RoboDK station: Station.rdk

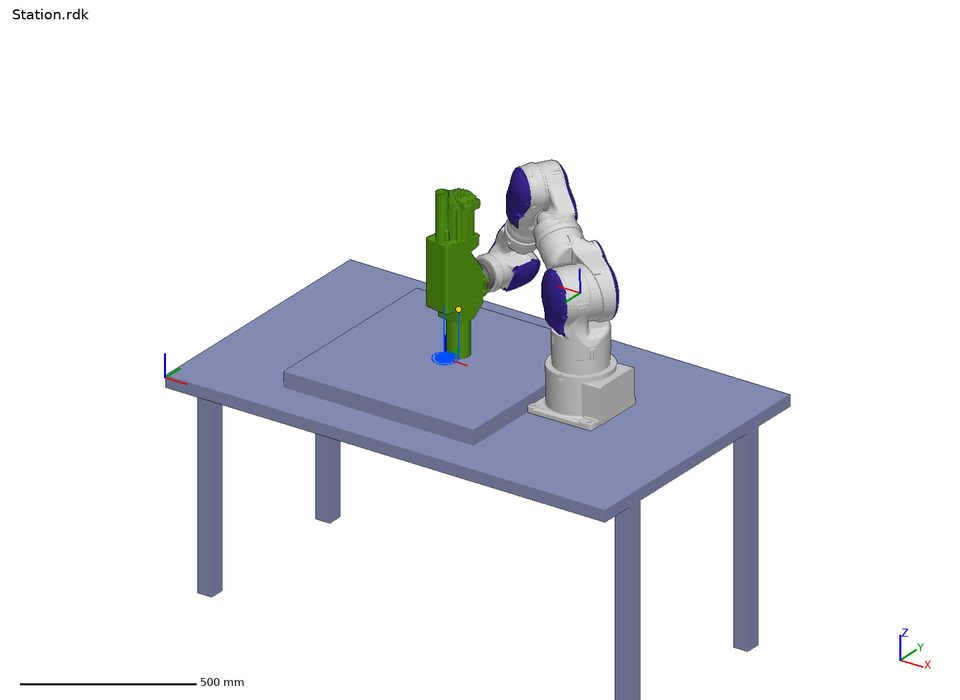
[picture v0: the station drawn from its stored meshes, robots at their saved joint values, targets as dots, program paths as lines]
Station Station (saved by RoboDK 5.5.3). Poses are relative to the parent item; angles as X-Y-Z fixed-axis rotations.
Station parameters (name, value as stored): Balls, 9000, lastSpeed, 40.0, LASTSPEED, 40.0
  - frame Yaskawa SIA10D Base at (1117.6, 457, 397.69) mm, rotated rx 0 ry 0.65 rz -180 deg
    - robot Yaskawa SIA10D: 7 axes, payload 10 kg, reach 720 mm, repeatability 0.1 mm, weight 60 kg
        modified DH rows (alpha deg, a mm, theta deg, d mm): 0, 0, 0, 360; -90, 0, 0, 0; 90, 0, 0, 360; -90, 0, 0, 0; 90, 0, 0, 360; -90, 0, 0, 0; 90, 0, 180, 155
        base shift (0, 0, -360) mm
        joint limits [-180, -110, -170, -135, -180, -110, -180] to [180, 110, 170, 135, 180, 110, 180]; home [0, 0, 0, 90, 0, 0, 0]; saved at [-31.519, 54.462, 0, 96.238, 71.076, 100.442, -153.064]
      - tool MDPH2, TCP at (-228, 0, 70.1) mm, rotated rx 0 ry -90 rz 0 deg, size 541.9 x 124.6 x 162.8 mm, geometry from Working one.STEP
  - frame Printing Frame at (649.7, 457, 58.96) mm
    - object par3 at (0, 0, 0) mm, rotated rx 90 ry 0 rz 0 deg, size 59.1 x 2 x 60 mm, geometry from par3.STEP
  - machining project Print3D settings: C:/Users/ajh269/AppData/Local/Temp/par2.stl | rotZ(0) | rotX(0)*rotY(0) | rotz(0)
  - Python program MCodeHandler (listed below)
  - Python program onStart (listed below)
  - Python program ExtruderHandler (listed below)
  - object table at (0, 0, -30) mm, rotated rx 90 ry 0 rz 0 deg, size 1524 x 739.1 x 914.4 mm, geometry from table.STEP
  - frame Table Corner at (0, 0, 0) mm
  - object MD_Bed at (320.1, 127, 5.56) mm, rotated rx 90 ry 0 rz 180 deg, size 660 x 53.3 x 660 mm, geometry from MD_Bed.STEP
  - machining project Print3D settings: C:/Users/ajh269/AppData/Local/Temp/par3.stl | rotZ(0) | rotX(0)*rotY(0) | rotz(0) | onStart | onPathStart | onApproach | onPoint | onRetract | onFinish | SetRPM(%1) | SetTool(%1) | ExtruderHandler(%1) | default | default | OutOnMov(%1) | OutOffMov(%1) | onPathFinish | MCodeHandler(%1)
  - program Print3D (604 instructions, listed below)
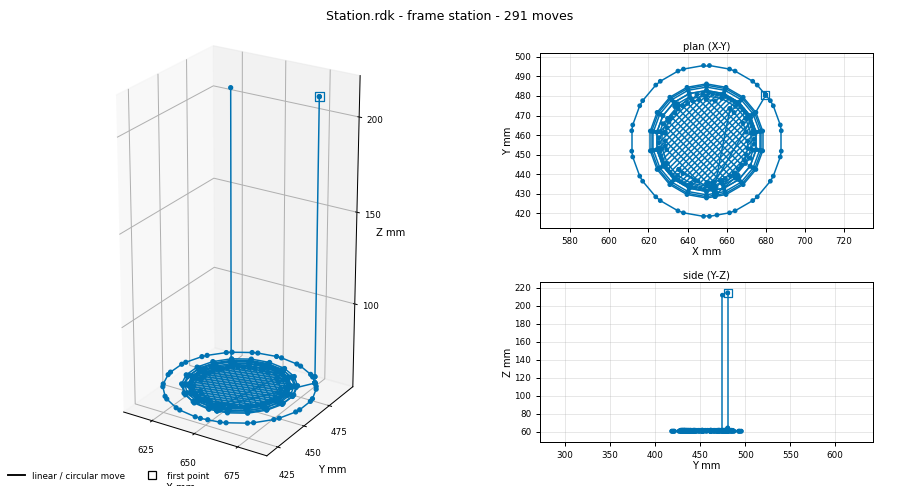
[picture p0: tool path of Station.rdk in frame station, 291 of 291 moves have a stored position in this frame; points joined in program order, loops and branches not executed]

--- Python program MCodeHandler ---
import sys

def handleFanOn():
    pass

def handleFanOff():
    pass

def handleTemperatureAsync():
    pass

def handleTemperatureSync():
    pass

# Create a mapping for the instruction codes
callbacks = {
    106: handleFanOn,
    107: handleFanOff,
    104: handleTemperatureAsync,
    109: handleTemperatureSync,
}

if len(sys.argv) > 1:
    instructionCode = int(sys.argv[1])
    print(instructionCode)

    if(len(sys.argv) > 2):
        arg = float(sys.argv[2])
        print(arg)

    #check for a second argument depending on the first

# Provoking an exception will display the console output if you run this script from RoboDK
# raise Exception('Display output. If program was run accidentally, move the error message above the pause button on RoboDK and click fast. (Shortcut is Backspace)')

--- Python program onStart ---
# import serial

# ser = serial.Serial('COM6', 9600, timeout=1.0)

# ser.write(b"NEW_PRINT\n")
# print(ser.readline())

--- Python program ExtruderHandler ---
# Type help("robodk.robolink") or help("robodk.robomath") for more information
# Press F5 to run the script
# Documentation: https://robodk.com/doc/en/RoboDK-API.html
# Reference:     https://robodk.com/doc/en/PythonAPI/robodk.html
# Note: It is not required to keep a copy of this file, your Python script is saved with your RDK project

# You can also use the new version of the API:
# from robodk import robolink    # RoboDK API
# from robodk import robomath    # Robot toolbox
# RDK = robolink.Robolink()

# Forward and backwards compatible use of the RoboDK API:
# Remove these 2 lines to follow python programming guidelines
# from robodk import *      # RoboDK API
# from robolink import *    # Robot toolbox
# Link to RoboDK
# RDK = Robolink()

import socket

message = b'{ distance: %f, materialLength: %f, newSpeed: %f }' % (1, 1, 0)

UDP_IP = "10.0.0.111"
UDP_PORT = 8888

sock = socket.socket(socket.AF_INET, # Internet
                    socket.SOCK_DGRAM) # UDP
sock.sendto(message, (UDP_IP, UDP_PORT))

# Provoking an exception will display the console output if you run this script from RoboDK
# raise Exception('Display output. If program was run accidentally, move the error message above the pause button on RoboDK and click fast. (Shortcut is Backspace)')

--- program Print3D (robot Yaskawa SIA10D) ---
  Smooth(1)
  Call MCodeHandler(107)
  Call MCodeHandler(104)
  Set speed (83.3 mm/s)
  Set Ref.: Printing Frame
  Set Tool: MDPH2
  Show MDPH2
  MoveJ 1 to (30.12, 23.57, 155) mm, rotated rx 180 ry 0 rz -100 deg; joints [-31.631, 34.814, 0, 98.46, 74.874, 105.649, -135.983]
  MoveL 2 to (30.12, 23.57, 155) mm, rotated rx 180 ry 0 rz -100 deg; joints [-31.631, 34.814, 0, 98.46, 74.874, 105.649, -135.983]
  MoveL 3 to (30.12, 23.57, 5) mm, rotated rx 180 ry 0 rz -100 deg; joints [-31.522, 53.972, 0, 96.405, 71.131, 100.548, -152.753]
  MoveL 4 to (30.12, 23.57, 5) mm, rotated rx 180 ry 0 rz -100 deg; joints [-31.522, 53.972, 0, 96.405, 71.131, 100.548, -152.753]
  Call MCodeHandler(109)
  Call MCodeHandler(83)
  Set speed (130.0 mm/s)
  MoveL 5 to (30.12, 23.57, 1.5) mm, rotated rx 180 ry 0 rz -100 deg; joints [-31.519, 54.462, 0, 96.238, 71.076, 100.442, -153.064]
  Call ExtruderHandler(-14.137...: ExtruderHandler(-14.13717)
  Set speed (40.0 mm/s)
  MoveL 6 to (30.12, 23.57, 1.5) mm, rotated rx 180 ry 0 rz -100 deg; joints [-31.519, 54.462, 0, 96.238, 71.076, 100.442, -153.064]
  Set speed (130.0 mm/s)
  MoveL 7 to (30.12, 23.57, 1.5) mm, rotated rx 180 ry 0 rz -100 deg; joints [-31.519, 54.462, 0, 96.238, 71.076, 100.442, -153.064]
  Call ExtruderHandler(14.13717)
  Set speed (40.0 mm/s)
  MoveL 8 to (30.12, 23.57, 1.5) mm, rotated rx 180 ry 0 rz -100 deg; joints [-31.519, 54.462, 0, 96.238, 71.076, 100.442, -153.064]
  Set speed (30.0 mm/s)
  MoveL 9 to (30.12, 23.57, 1.5) mm, rotated rx 180 ry 0 rz -100 deg; joints [-31.519, 54.462, 0, 96.238, 71.076, 100.442, -153.064]
  Call ExtruderHandler(26.15888)
  MoveL 10 to (25.93, 28.56, 1.5) mm, rotated rx -180 ry 0 rz -100 deg; joints [-31.768, 54.946, 0, 94.943, 70.997, 100.822, -152.324]
  Call ExtruderHandler(12.10715)
  MoveL 11 to (23.62, 30.5, 1.5) mm, rotated rx -180 ry 0 rz -100 deg; joints [-31.82, 55.182, 0, 94.314, 71.022, 100.974, -151.954]
  Call ExtruderHandler(41.85421)
  MoveL 12 to (14.6, 35.71, 1.5) mm, rotated rx -180 ry 0 rz -100 deg; joints [-31.781, 56.028, 0, 92.089, 71.315, 101.401, -150.617]
  Call ExtruderHandler(12.10718)
  MoveL 13 to (11.77, 36.74, 1.5) mm, rotated rx -180 ry 0 rz -100 deg; joints [-31.71, 56.273, 0, 91.451, 71.453, 101.49, -150.225]
  Call ExtruderHandler(41.85419)
  MoveL 14 to (1.51, 38.55, 1.5) mm, rotated rx 180 ry 0 rz -100 deg; joints [-31.269, 57.096, 0, 89.328, 72.091, 101.669, -148.889]
  Call ExtruderHandler(12.10714)
  MoveL 15 to (-1.51, 38.55, 1.5) mm, rotated rx 180 ry 0 rz -100 deg; joints [-31.091, 57.32, 0, 88.757, 72.314, 101.681, -148.519]
  Call ExtruderHandler(41.85422)
  MoveL 16 to (-11.77, 36.74, 1.5) mm, rotated rx -180 ry 0 rz -100 deg; joints [-30.325, 58.016, 0, 86.988, 73.183, 101.585, -147.342]
  Call ExtruderHandler(12.10717)
  MoveL 17 to (-14.6, 35.71, 1.5) mm, rotated rx -180 ry 0 rz -100 deg; joints [-30.066, 58.189, 0, 86.551, 73.455, 101.518, -147.041]
  Call ExtruderHandler(41.85421)
  MoveL 18 to (-23.62, 30.5, 1.5) mm, rotated rx 180 ry 0 rz -100 deg; joints [-29.069, 58.666, 0, 85.348, 74.438, 101.161, -146.165]
  Call ExtruderHandler(12.10715)
  MoveL 19 to (-25.93, 28.56, 1.5) mm, rotated rx 180 ry 0 rz -100 deg; joints [-28.759, 58.765, 0, 85.099, 74.726, 101.025, -145.968]
  Call ExtruderHandler(41.85420)
  MoveL 20 to (-32.63, 20.58, 1.5) mm, rotated rx 180 ry 0 rz -100 deg; joints [-27.638, 58.956, 0, 84.61, 75.717, 100.46, -145.503]
  Call ExtruderHandler(12.10718)
  MoveL 21 to (-34.14, 17.97, 1.5) mm, rotated rx 180 ry 0 rz -100 deg; joints [-27.308, 58.967, 0, 84.58, 75.995, 100.274, -145.435]
  Call ExtruderHandler(41.85421)
  MoveL 22 to (-37.7, 8.18, 1.5) mm, rotated rx 180 ry 0 rz -100 deg; joints [-26.172, 58.846, 0, 84.865, 76.909, 99.581, -145.437]
  Call ExtruderHandler(12.10715)
  MoveL 23 to (-38.22, 5.21, 1.5) mm, rotated rx -180 ry 0 rz -100 deg; joints [-25.853, 58.766, 0, 85.058, 77.155, 99.372, -145.506]
  Call ExtruderHandler(41.85420)
  MoveL 24 to (-38.22, -5.21, 1.5) mm, rotated rx -180 ry 0 rz -100 deg; joints [-24.811, 58.349, 0, 86.082, 77.926, 98.645, -145.973]
  Call ExtruderHandler(12.10715)
  MoveL 25 to (-37.7, -8.18, 1.5) mm, rotated rx 180 ry 0 rz -100 deg; joints [-24.535, 58.192, 0, 86.473, 78.121, 98.44, -146.17]
  Call ExtruderHandler(41.85422)
  MoveL 26 to (-34.14, -17.97, 1.5) mm, rotated rx 180 ry 0 rz -100 deg; joints [-23.696, 57.537, 0, 88.11, 78.687, 97.773, -147.044]
  Call ExtruderHandler(12.10716)
  MoveL 27 to (-32.63, -20.58, 1.5) mm, rotated rx -180 ry 0 rz -100 deg; joints [-23.493, 57.322, 0, 88.651, 78.814, 97.597, -147.345]
  Call ExtruderHandler(41.85420)
  MoveL 28 to (-25.93, -28.56, 1.5) mm, rotated rx -180 ry 0 rz -80 deg; joints [-19.878, 63.594, 0, 73.405, 67.135, 109.774, -141.706]
  Call ExtruderHandler(12.10716)
  MoveL 29 to (-23.62, -30.5, 1.5) mm, rotated rx 180 ry 0 rz -80 deg; joints [-19.773, 63.278, 0, 74.141, 67.083, 109.544, -142.089]
  Call ExtruderHandler(41.85421)
  MoveL 30 to (-14.6, -35.71, 1.5) mm, rotated rx 180 ry 0 rz -80 deg; joints [-19.582, 62.167, 0, 76.758, 66.761, 108.837, -143.502]
  Call ExtruderHandler(12.10716)
  MoveL 31 to (-11.77, -36.74, 1.5) mm, rotated rx 180 ry 0 rz -80 deg; joints [-19.58, 61.849, 0, 77.513, 66.626, 108.662, -143.926]
  Call ExtruderHandler(41.85420)
  MoveL 32 to (-1.51, -38.55, 1.5) mm, rotated rx -180 ry 0 rz -80 deg; joints [-19.763, 60.795, 0, 80.039, 66.021, 108.179, -145.395]
  Call ExtruderHandler(12.10714)
  MoveL 33 to (1.51, -38.55, 1.5) mm, rotated rx 180 ry 0 rz -80 deg; joints [-19.872, 60.511, 0, 80.724, 65.808, 108.078, -145.811]
  Call ExtruderHandler(15.69532)
  MoveL 34 to (5.36, -37.87, 1.5) mm, rotated rx -180 ry 0 rz -80 deg; joints [-20.08, 60.177, 0, 81.535, 65.486, 107.999, -146.324]
  Call ExtruderHandler(26.15890)
  MoveL 35 to (11.77, -36.74, 1.5) mm, rotated rx 180 ry 0 rz -80 deg; joints [-20.433, 59.631, 0, 82.869, 64.946, 107.866, -147.171]
  Call ExtruderHandler(12.10714)
  MoveL 36 to (14.6, -35.71, 1.5) mm, rotated rx 180 ry 0 rz -80 deg; joints [-20.645, 59.413, 0, 83.406, 64.667, 107.846, -147.532]
  Call ExtruderHandler(41.85423)
  MoveL 37 to (23.62, -30.5, 1.5) mm, rotated rx 180 ry 0 rz -80 deg; joints [-21.531, 58.8, 0, 84.926, 63.619, 107.928, -148.632]
  Call ExtruderHandler(12.10716)
  MoveL 38 to (25.93, -28.56, 1.5) mm, rotated rx 180 ry 0 rz -80 deg; joints [-21.823, 58.668, 0, 85.255, 63.301, 107.994, -148.899]
  Call ExtruderHandler(41.85420)
  MoveL 39 to (32.63, -20.58, 1.5) mm, rotated rx 180 ry 0 rz -80 deg; joints [-22.922, 58.383, 0, 85.976, 62.186, 108.366, -149.617]
  Call ExtruderHandler(12.10714)
  MoveL 40 to (34.14, -17.97, 1.5) mm, rotated rx -180 ry 0 rz -80 deg; joints [-23.254, 58.352, 0, 86.058, 61.871, 108.513, -149.76]
  Call ExtruderHandler(41.85421)
  MoveL 41 to (37.7, -8.18, 1.5) mm, rotated rx 180 ry 0 rz -80 deg; joints [-24.408, 58.422, 0, 85.897, 60.851, 109.147, -150.015]
  Call ExtruderHandler(12.10718)
  MoveL 42 to (38.22, -5.21, 1.5) mm, rotated rx 180 ry 0 rz -80 deg; joints [-24.731, 58.493, 0, 85.723, 60.588, 109.362, -150.018]
  Call ExtruderHandler(41.85420)
  MoveL 43 to (38.22, 5.21, 1.5) mm, rotated rx -180 ry 0 rz -100 deg; joints [-30.075, 53.231, 0, 99.601, 72.038, 99.119, -154.896]
  Call ExtruderHandler(12.10718)
  MoveL 44 to (37.7, 8.18, 1.5) mm, rotated rx 180 ry 0 rz -100 deg; joints [-30.365, 53.375, 0, 99.205, 71.812, 99.324, -154.695]
  Call ExtruderHandler(41.85422)
  MoveL 45 to (34.14, 17.97, 1.5) mm, rotated rx -180 ry 0 rz -100 deg; joints [-31.188, 53.977, 0, 97.553, 71.234, 100.022, -153.809]
  Call ExtruderHandler(12.10713)
  MoveL 46 to (32.63, 20.58, 1.5) mm, rotated rx 180 ry 0 rz -100 deg; joints [-31.367, 54.178, 0, 97.007, 71.131, 100.215, -153.506]
  Call ExtruderHandler(14.79146)
  MoveL 47 to (30.26, 23.4, 1.5) mm, rotated rx 180 ry 0 rz -100 deg; joints [-31.511, 54.446, 0, 96.282, 71.079, 100.429, -153.089]
  Call ExtruderHandler(-14.137...: ExtruderHandler(-14.13717)
  Set speed (40.0 mm/s)
  MoveL 48 to (30.26, 23.4, 1.5) mm, rotated rx 180 ry 0 rz -100 deg; joints [-31.511, 54.446, 0, 96.282, 71.079, 100.429, -153.089]
  Set speed (130.0 mm/s)
  MoveL 49 to (3.4, -22.44, 1.5) mm, rotated rx -180 ry 0 rz -80 deg; joints [-21.539, 60.913, 0, 79.77, 64.533, 109.262, -145.748]
  Call ExtruderHandler(14.13717)
  Set speed (40.0 mm/s)
  MoveL 50 to (3.4, -22.44, 1.5) mm, rotated rx -180 ry 0 rz -80 deg; joints [-21.539, 60.913, 0, 79.77, 64.533, 109.262, -145.748]
  Set speed (30.0 mm/s)
  MoveL 51 to (3.4, -22.44, 1.5) mm, rotated rx -180 ry 0 rz -80 deg; joints [-21.539, 60.913, 0, 79.77, 64.533, 109.262, -145.748]
  Call ExtruderHandler(18.28870)
  MoveL 52 to (7.88, -21.65, 1.5) mm, rotated rx -180 ry 0 rz -80 deg; joints [-21.792, 60.526, 0, 80.708, 64.139, 109.168, -146.346]
  Call ExtruderHandler(32.14129)
  MoveL 53 to (14.81, -17.65, 1.5) mm, rotated rx 180 ry 0 rz -80 deg; joints [-22.467, 60.044, 0, 81.882, 63.33, 109.237, -147.2]
  Call ExtruderHandler(32.14129)
  MoveL 54 to (19.95, -11.52, 1.5) mm, rotated rx 180 ry 0 rz -80 deg; joints [-23.289, 59.819, 0, 82.44, 62.496, 109.536, -147.758]
  Call ExtruderHandler(32.14130)
  MoveL 55 to (22.69, -4, 1.5) mm, rotated rx 180 ry 0 rz -100 deg; joints [-28.12, 53.888, 0, 97.749, 73.988, 98.597, -153.471]
  Call ExtruderHandler(32.14128)
  MoveL 56 to (22.69, 4, 1.5) mm, rotated rx 180 ry 0 rz -100 deg; joints [-28.988, 54.182, 0, 96.958, 73.281, 99.136, -153.107]
  Call ExtruderHandler(32.14131)
  MoveL 57 to (19.95, 11.52, 1.5) mm, rotated rx 180 ry 0 rz -100 deg; joints [-29.626, 54.653, 0, 95.695, 72.836, 99.665, -152.43]
  Call ExtruderHandler(32.14129)
  MoveL 58 to (14.81, 17.65, 1.5) mm, rotated rx 180 ry 0 rz -100 deg; joints [-29.959, 55.247, 0, 94.113, 72.703, 100.117, -151.523]
  Call ExtruderHandler(32.14130)
  MoveL 59 to (7.88, 21.65, 1.5) mm, rotated rx 180 ry 0 rz -100 deg; joints [-29.96, 55.897, 0, 92.405, 72.886, 100.431, -150.495]
  Call ExtruderHandler(32.14128)
  MoveL 60 to (0, 23.04, 1.5) mm, rotated rx 180 ry 0 rz -100 deg; joints [-29.643, 56.523, 0, 90.774, 73.341, 100.561, -149.468]
  Call ExtruderHandler(32.14129)
  MoveL 61 to (-7.88, 21.65, 1.5) mm, rotated rx 180 ry 0 rz -100 deg; joints [-29.06, 57.049, 0, 89.417, 73.995, 100.489, -148.566]
  Call ExtruderHandler(32.14130)
  MoveL 62 to (-14.81, 17.65, 1.5) mm, rotated rx 180 ry 0 rz -100 deg; joints [-28.281, 57.407, 0, 88.495, 74.762, 100.224, -147.895]
  Call ExtruderHandler(32.14129)
  MoveL 63 to (-19.95, 11.52, 1.5) mm, rotated rx 180 ry 0 rz -100 deg; joints [-27.395, 57.551, 0, 88.12, 75.556, 99.801, -147.539]
  Call ExtruderHandler(32.14129)
  MoveL 64 to (-22.69, 4, 1.5) mm, rotated rx 180 ry 0 rz -100 deg; joints [-26.497, 57.46, 0, 88.339, 76.299, 99.28, -147.539]
  Call ExtruderHandler(32.14129)
  MoveL 65 to (-22.69, -4, 1.5) mm, rotated rx -180 ry 0 rz -100 deg; joints [-25.68, 57.147, 0, 89.123, 76.921, 98.726, -147.896]
  Call ExtruderHandler(32.14129)
  MoveL 66 to (-19.95, -11.52, 1.5) mm, rotated rx -180 ry 0 rz -100 deg; joints [-25.035, 56.653, 0, 90.378, 77.361, 98.211, -148.567]
  Call ExtruderHandler(32.14129)
  MoveL 67 to (-14.81, -17.65, 1.5) mm, rotated rx -180 ry 0 rz -100 deg; joints [-24.64, 56.041, 0, 91.955, 77.568, 97.795, -149.472]
  Call ExtruderHandler(32.14130)
  MoveL 68 to (-7.88, -21.65, 1.5) mm, rotated rx -180 ry 0 rz -80 deg; joints [-21.186, 62.026, 0, 77.108, 65.333, 109.713, -144.157]
  Call ExtruderHandler(32.14129)
  MoveL 69 to (0, -23.04, 1.5) mm, rotated rx 180 ry 0 rz -80 deg; joints [-21.349, 61.212, 0, 79.052, 64.83, 109.333, -145.291]
  Call ExtruderHandler(12.94872)
  MoveL 70 to (3.17, -22.48, 1.5) mm, rotated rx 180 ry 0 rz -80 deg; joints [-21.526, 60.933, 0, 79.723, 64.552, 109.267, -145.718]
  Call ExtruderHandler(-14.137...: ExtruderHandler(-14.13717)
  Set speed (40.0 mm/s)
  MoveL 71 to (3.17, -22.48, 1.5) mm, rotated rx 180 ry 0 rz -80 deg; joints [-21.526, 60.933, 0, 79.723, 64.552, 109.267, -145.718]
  Set speed (130.0 mm/s)
  MoveL 72 to (3.86, -25.08, 1.5) mm, rotated rx 180 ry 0 rz -80 deg; joints [-21.297, 60.771, 0, 80.11, 64.681, 109.04, -145.867]
  Call ExtruderHandler(14.13717)
  Set speed (40.0 mm/s)
  MoveL 73 to (3.86, -25.08, 1.5) mm, rotated rx 180 ry 0 rz -80 deg; joints [-21.297, 60.771, 0, 80.11, 64.681, 109.04, -145.867]
  Set speed (30.0 mm/s)
  MoveL 74 to (3.86, -25.08, 1.5) mm, rotated rx 180 ry 0 rz -80 deg; joints [-21.297, 60.771, 0, 80.11, 64.681, 109.04, -145.867]
  Call ExtruderHandler(20.18568)
  MoveL 75 to (8.81, -24.2, 1.5) mm, rotated rx 180 ry 0 rz -80 deg; joints [-21.576, 60.345, 0, 81.143, 64.249, 108.936, -146.526]
  Call ExtruderHandler(35.93525)
  MoveL 76 to (16.56, -19.73, 1.5) mm, rotated rx 180 ry 0 rz -80 deg; joints [-22.331, 59.809, 0, 82.454, 63.345, 109.012, -147.479]
  Call ExtruderHandler(35.93525)
  MoveL 77 to (22.31, -12.88, 1.5) mm, rotated rx 180 ry 0 rz -80 deg; joints [-23.255, 59.558, 0, 83.076, 62.409, 109.343, -148.101]
  Call ExtruderHandler(35.93526)
  MoveL 78 to (25.37, -4.47, 1.5) mm, rotated rx 180 ry 0 rz -80 deg; joints [-24.221, 59.62, 0, 82.937, 61.567, 109.898, -148.321]
  Call ExtruderHandler(35.93524)
  MoveL 79 to (25.37, 4.47, 1.5) mm, rotated rx -180 ry 0 rz -100 deg; joints [-29.2, 54.024, 0, 97.394, 73.049, 99.153, -153.405]
  Call ExtruderHandler(35.93527)
  MoveL 80 to (22.31, 12.88, 1.5) mm, rotated rx 180 ry 0 rz -100 deg; joints [-29.912, 54.548, 0, 95.98, 72.55, 99.746, -152.648]
  Call ExtruderHandler(35.93524)
  MoveL 81 to (16.56, 19.73, 1.5) mm, rotated rx 180 ry 0 rz -100 deg; joints [-30.279, 55.212, 0, 94.212, 72.408, 100.254, -151.634]
  Call ExtruderHandler(35.93526)
  MoveL 82 to (8.81, 24.2, 1.5) mm, rotated rx 180 ry 0 rz -100 deg; joints [-30.274, 55.938, 0, 92.301, 72.62, 100.607, -150.485]
  Call ExtruderHandler(35.93524)
  MoveL 83 to (0, 25.76, 1.5) mm, rotated rx 180 ry 0 rz -100 deg; joints [-29.916, 56.64, 0, 90.478, 73.136, 100.754, -149.337]
  Call ExtruderHandler(35.93524)
  MoveL 84 to (-8.81, 24.2, 1.5) mm, rotated rx 180 ry 0 rz -100 deg; joints [-29.263, 57.229, 0, 88.96, 73.87, 100.673, -148.327]
  Call ExtruderHandler(35.93526)
  MoveL 85 to (-16.56, 19.73, 1.5) mm, rotated rx 180 ry 0 rz -100 deg; joints [-28.395, 57.631, 0, 87.93, 74.725, 100.375, -147.578]
  Call ExtruderHandler(35.93525)
  MoveL 86 to (-22.31, 12.88, 1.5) mm, rotated rx 180 ry 0 rz -100 deg; joints [-27.409, 57.792, 0, 87.511, 75.606, 99.901, -147.179]
  Call ExtruderHandler(35.93525)
  MoveL 87 to (-25.37, 4.47, 1.5) mm, rotated rx 180 ry 0 rz -100 deg; joints [-26.41, 57.69, 0, 87.755, 76.429, 99.315, -147.18]
  Call ExtruderHandler(35.93525)
  MoveL 88 to (-25.37, -4.47, 1.5) mm, rotated rx 180 ry 0 rz -100 deg; joints [-25.5, 57.339, 0, 88.632, 77.118, 98.696, -147.579]
  Call ExtruderHandler(35.93525)
  MoveL 89 to (-22.31, -12.88, 1.5) mm, rotated rx 180 ry 0 rz -100 deg; joints [-24.779, 56.785, 0, 90.036, 77.609, 98.12, -148.329]
  Call ExtruderHandler(35.93525)
  MoveL 90 to (-16.56, -19.73, 1.5) mm, rotated rx 180 ry 0 rz -100 deg; joints [-24.333, 56.1, 0, 91.798, 77.846, 97.657, -149.34]
  Call ExtruderHandler(35.93526)
  MoveL 91 to (-8.81, -24.2, 1.5) mm, rotated rx -180 ry 0 rz -80 deg; joints [-20.905, 62.02, 0, 77.121, 65.571, 109.543, -144.082]
  Call ExtruderHandler(35.93525)
  MoveL 92 to (0, -25.76, 1.5) mm, rotated rx 180 ry 0 rz -80 deg; joints [-21.083, 61.11, 0, 79.293, 65.016, 109.12, -145.349]
  Call ExtruderHandler(14.84570)
  MoveL 93 to (3.64, -25.12, 1.5) mm, rotated rx 180 ry 0 rz -80 deg; joints [-21.285, 60.791, 0, 80.063, 64.7, 109.044, -145.837]
  Call ExtruderHandler(-14.137...: ExtruderHandler(-14.13717)
  Set speed (40.0 mm/s)
  MoveL 94 to (3.64, -25.12, 1.5) mm, rotated rx 180 ry 0 rz -80 deg; joints [-21.285, 60.791, 0, 80.063, 64.7, 109.044, -145.837]
  Set speed (130.0 mm/s)
  MoveL 95 to (4.33, -27.71, 1.5) mm, rotated rx -180 ry 0 rz -80 deg; joints [-21.054, 60.631, 0, 80.446, 64.831, 108.818, -145.985]
  Call ExtruderHandler(14.13717)
  Set speed (40.0 mm/s)
  MoveL 96 to (4.33, -27.71, 1.5) mm, rotated rx -180 ry 0 rz -80 deg; joints [-21.054, 60.631, 0, 80.446, 64.831, 108.818, -145.985]
  Set speed (30.0 mm/s)
  MoveL 97 to (4.33, -27.71, 1.5) mm, rotated rx -180 ry 0 rz -80 deg; joints [-21.054, 60.631, 0, 80.446, 64.831, 108.818, -145.985]
  Call ExtruderHandler(22.08266)
  MoveL 98 to (9.74, -26.76, 1.5) mm, rotated rx 180 ry 0 rz -80 deg; joints [-21.358, 60.166, 0, 81.574, 64.363, 108.704, -146.704]
  Call ExtruderHandler(39.72921)
  MoveL 99 to (18.3, -21.82, 1.5) mm, rotated rx 180 ry 0 rz -80 deg; joints [-22.194, 59.576, 0, 83.022, 63.364, 108.787, -147.756]
  Call ExtruderHandler(39.72921)
  MoveL 100 to (24.66, -14.24, 1.5) mm, rotated rx -180 ry 0 rz -80 deg; joints [-23.22, 59.3, 0, 83.709, 62.324, 109.151, -148.442]
  Call ExtruderHandler(39.72921)
  MoveL 101 to (28.04, -4.95, 1.5) mm, rotated rx 180 ry 0 rz -80 deg; joints [-24.294, 59.368, 0, 83.555, 61.386, 109.762, -148.685]
  Call ExtruderHandler(39.72921)
  MoveL 102 to (28.04, 4.95, 1.5) mm, rotated rx -180 ry 0 rz -100 deg; joints [-29.413, 53.867, 0, 97.826, 72.814, 99.169, -153.703]
  Call ExtruderHandler(39.72922)
  MoveL 103 to (24.66, 14.24, 1.5) mm, rotated rx 180 ry 0 rz -100 deg; joints [-30.199, 54.446, 0, 96.262, 72.263, 99.826, -152.865]
  Call ExtruderHandler(39.72920)
  MoveL 104 to (18.31, 21.81, 1.5) mm, rotated rx 180 ry 0 rz -100 deg; joints [-30.601, 55.178, 0, 94.306, 72.112, 100.391, -151.744]
  Call ExtruderHandler(39.72922)
  MoveL 105 to (9.74, 26.76, 1.5) mm, rotated rx 180 ry 0 rz -100 deg; joints [-30.588, 55.981, 0, 92.195, 72.356, 100.784, -150.473]
  Call ExtruderHandler(39.72920)
  MoveL 106 to (0, 28.48, 1.5) mm, rotated rx 180 ry 0 rz -100 deg; joints [-30.188, 56.757, 0, 90.179, 72.933, 100.949, -149.204]
  Call ExtruderHandler(39.72921)
  MoveL 107 to (-9.74, 26.76, 1.5) mm, rotated rx 180 ry 0 rz -100 deg; joints [-29.464, 57.411, 0, 88.501, 73.747, 100.859, -148.088]
  Call ExtruderHandler(39.72922)
  MoveL 108 to (-18.3, 21.81, 1.5) mm, rotated rx 180 ry 0 rz -100 deg; joints [-28.507, 57.858, 0, 87.361, 74.69, 100.527, -147.259]
  Call ExtruderHandler(39.72921)
  MoveL 109 to (-24.66, 14.24, 1.5) mm, rotated rx -180 ry 0 rz -100 deg; joints [-27.423, 58.036, 0, 86.898, 75.658, 100, -146.818]
  Call ExtruderHandler(39.72921)
  MoveL 110 to (-28.04, 4.94, 1.5) mm, rotated rx -180 ry 0 rz -100 deg; joints [-26.324, 57.923, 0, 87.168, 76.558, 99.35, -146.819]
  Call ExtruderHandler(39.72920)
  MoveL 111 to (-28.04, -4.95, 1.5) mm, rotated rx -180 ry 0 rz -100 deg; joints [-25.321, 57.533, 0, 88.138, 77.314, 98.664, -147.261]
  Call ExtruderHandler(39.72921)
  MoveL 112 to (-24.66, -14.24, 1.5) mm, rotated rx 180 ry 0 rz -100 deg; joints [-24.524, 56.919, 0, 89.69, 77.856, 98.029, -148.09]
  Call ExtruderHandler(39.72921)
  MoveL 113 to (-18.31, -21.81, 1.5) mm, rotated rx 180 ry 0 rz -100 deg; joints [-24.027, 56.16, 0, 91.638, 78.122, 97.518, -149.208]
  Call ExtruderHandler(39.72922)
  MoveL 114 to (-9.74, -26.76, 1.5) mm, rotated rx -180 ry 0 rz -80 deg; joints [-20.624, 62.014, 0, 77.13, 65.81, 109.374, -144.005]
  Call ExtruderHandler(39.72921)
  MoveL 115 to (0, -28.48, 1.5) mm, rotated rx 180 ry 0 rz -80 deg; joints [-20.816, 61.01, 0, 79.531, 65.204, 108.907, -145.405]
  Call ExtruderHandler(16.74268)
  MoveL 116 to (4.1, -27.75, 1.5) mm, rotated rx -180 ry 0 rz -80 deg; joints [-21.042, 60.65, 0, 80.399, 64.85, 108.822, -145.956]
  Set speed (130.0 mm/s)
  MoveL 117 to (4.84, -26.3, 1.5) mm, rotated rx 180 ry 0 rz -80 deg; joints [-21.213, 60.635, 0, 80.438, 64.694, 108.91, -146.027]
  Call ExtruderHandler(-14.137...: ExtruderHandler(-14.13717)
  Set speed (40.0 mm/s)
  MoveL 118 to (4.84, -26.3, 1.5) mm, rotated rx 180 ry 0 rz -80 deg; joints [-21.213, 60.635, 0, 80.438, 64.694, 108.91, -146.027]
  Set speed (130.0 mm/s)
  MoveL 119 to (-14.1, -14.52, 1.5) mm, rotated rx 180 ry 0 rz -100 deg; joints [-25.006, 56.099, 0, 91.809, 77.264, 98.004, -149.428]
  Call ExtruderHandler(14.13717)
  Set speed (40.0 mm/s)
  MoveL 120 to (-14.1, -14.52, 1.5) mm, rotated rx -180 ry 0 rz -100 deg; joints [-25.006, 56.099, 0, 91.809, 77.264, 98.004, -149.428]
  Set speed (30.0 mm/s)
  MoveL 121 to (-14.1, -14.52, 1.5) mm, rotated rx -180 ry 0 rz -100 deg; joints [-25.006, 56.099, 0, 91.809, 77.264, 98.004, -149.428]
  Call ExtruderHandler(11.92574)
  MoveL 122 to (-12.02, -16.61, 1.5) mm, rotated rx 180 ry 0 rz -100 deg; joints [-24.888, 55.869, 0, 92.406, 77.316, 97.862, -149.776]
  Call ExtruderHandler(28.56512)
  MoveL 123 to (-5.91, -20.13, 1.5) mm, rotated rx -180 ry 0 rz -80 deg; joints [-21.407, 61.892, 0, 77.429, 65.084, 109.765, -144.401]
  Call ExtruderHandler(6.15843)
  MoveL 124 to (-4.41, -20.4, 1.5) mm, rotated rx 180 ry 0 rz -80 deg; joints [-21.438, 61.736, 0, 77.8, 64.987, 109.693, -144.618]
  Call ExtruderHandler(91.11342)
  MoveL 125 to (-20.32, -4.48, 1.5) mm, rotated rx -180 ry 0 rz -100 deg; joints [-25.747, 56.944, 0, 89.64, 76.816, 98.691, -148.215]
  Call ExtruderHandler(8.60510)
  MoveL 126 to (-21.05, -2.49, 1.5) mm, rotated rx 180 ry 0 rz -100 deg; joints [-25.917, 57.077, 0, 89.303, 76.702, 98.829, -148.036]
  Call ExtruderHandler(10.30798)
  MoveL 127 to (-21.05, 0.06, 1.5) mm, rotated rx 180 ry 0 rz -100 deg; joints [-26.178, 57.176, 0, 89.055, 76.502, 99.005, -147.922]
  Call ExtruderHandler(121.804...: ExtruderHandler(121.80441)
  MoveL 128 to (0.22, -21.22, 1.5) mm, rotated rx 180 ry 0 rz -80 deg; joints [-21.536, 61.26, 0, 78.939, 64.689, 109.468, -145.283]
  Call ExtruderHandler(3.36032)
  MoveL 129 to (1.04, -21.36, 1.5) mm, rotated rx 180 ry 0 rz -80 deg; joints [-21.554, 61.176, 0, 79.139, 64.637, 109.429, -145.399]
  Call ExtruderHandler(10.98469)
  MoveL 130 to (3.71, -20.89, 1.5) mm, rotated rx -180 ry 0 rz -80 deg; joints [-21.703, 60.942, 0, 79.703, 64.402, 109.373, -145.758]
  Call ExtruderHandler(141.783...: ExtruderHandler(141.78311)
  MoveL 131 to (-21.05, 3.88, 1.5) mm, rotated rx 180 ry 0 rz -100 deg; joints [-26.567, 57.326, 0, 88.677, 76.207, 99.269, -147.751]
  Call ExtruderHandler(2.80780)
  MoveL 132 to (-21.05, 4.57, 1.5) mm, rotated rx 180 ry 0 rz -100 deg; joints [-26.638, 57.354, 0, 88.608, 76.153, 99.317, -147.719]
  Call ExtruderHandler(9.86432)
  MoveL 133 to (-20.22, 6.86, 1.5) mm, rotated rx 180 ry 0 rz -100 deg; joints [-26.912, 57.381, 0, 88.543, 75.926, 99.476, -147.72]
  Call ExtruderHandler(155.587...: ExtruderHandler(155.58748)
  MoveL 134 to (6.96, -20.32, 1.5) mm, rotated rx 180 ry 0 rz -80 deg; joints [-21.887, 60.661, 0, 80.382, 64.116, 109.305, -146.191]
  Call ExtruderHandler(4.24451)
  MoveL 135 to (7.99, -20.14, 1.5) mm, rotated rx 180 ry 0 rz -80 deg; joints [-21.946, 60.572, 0, 80.596, 64.025, 109.283, -146.329]
  Call ExtruderHandler(7.71138)
  MoveL 136 to (9.64, -19.18, 1.5) mm, rotated rx 180 ry 0 rz -80 deg; joints [-22.106, 60.456, 0, 80.878, 63.833, 109.3, -146.533]
  Call ExtruderHandler(165.112...: ExtruderHandler(165.11256)
  MoveL 137 to (-19.2, 9.66, 1.5) mm, rotated rx -180 ry 0 rz -100 deg; joints [-27.247, 57.415, 0, 88.461, 75.648, 99.67, -147.719]
  Call ExtruderHandler(6.64751)
  MoveL 138 to (-18.64, 11.2, 1.5) mm, rotated rx 180 ry 0 rz -100 deg; joints [-27.432, 57.435, 0, 88.414, 75.496, 99.777, -147.718]
  Call ExtruderHandler(4.91956)
  MoveL 139 to (-17.86, 12.13, 1.5) mm, rotated rx -180 ry 0 rz -100 deg; joints [-27.566, 57.413, 0, 88.472, 75.375, 99.841, -147.773]
  Call ExtruderHandler(171.278...: ExtruderHandler(171.27818)
  MoveL 140 to (12.06, -17.79, 1.5) mm, rotated rx 180 ry 0 rz -80 deg; joints [-22.341, 60.288, 0, 81.288, 63.55, 109.324, -146.832]
  Call ExtruderHandler(9.54450)
  MoveL 141 to (14.1, -16.61, 1.5) mm, rotated rx 180 ry 0 rz -80 deg; joints [-22.541, 60.148, 0, 81.632, 63.31, 109.344, -147.083]
  Call ExtruderHandler(1.71277)
  MoveL 142 to (14.37, -16.28, 1.5) mm, rotated rx 180 ry 0 rz -80 deg; joints [-22.584, 60.135, 0, 81.662, 63.266, 109.36, -147.112]
  Call ExtruderHandler(174.555...: ExtruderHandler(174.55505)
  MoveL 143 to (-16.12, 14.21, 1.5) mm, rotated rx 180 ry 0 rz -100 deg; joints [-27.867, 57.364, 0, 88.6, 75.105, 99.983, -147.894]
  Call ExtruderHandler(10.96726)
  MoveL 144 to (-14.37, 16.28, 1.5) mm, rotated rx -180 ry 0 rz -100 deg; joints [-28.168, 57.316, 0, 88.724, 74.835, 100.126, -148.014]
  Call ExtruderHandler(174.555...: ExtruderHandler(174.55505)
  MoveL 145 to (16.11, -14.21, 1.5) mm, rotated rx 180 ry 0 rz -80 deg; joints [-22.861, 60.058, 0, 81.853, 62.985, 109.461, -147.302]
  Call ExtruderHandler(10.96725)
  MoveL 146 to (17.86, -12.13, 1.5) mm, rotated rx -180 ry 0 rz -80 deg; joints [-23.14, 59.982, 0, 82.041, 62.703, 109.563, -147.491]
  Call ExtruderHandler(171.278...: ExtruderHandler(171.27816)
  MoveL 147 to (-12.06, 17.78, 1.5) mm, rotated rx 180 ry 0 rz -100 deg; joints [-28.443, 57.202, 0, 89.018, 74.568, 100.227, -148.231]
  Call ExtruderHandler(11.31093)
  MoveL 148 to (-9.64, 19.18, 1.5) mm, rotated rx 180 ry 0 rz -100 deg; joints [-28.715, 57.077, 0, 89.34, 74.3, 100.319, -148.465]
  Call ExtruderHandler(165.112...: ExtruderHandler(165.11255)
  MoveL 149 to (19.2, -9.66, 1.5) mm, rotated rx -180 ry 0 rz -80 deg; joints [-23.441, 59.959, 0, 82.101, 62.423, 109.71, -147.616]
  Call ExtruderHandler(12.05498)
  MoveL 150 to (20.22, -6.86, 1.5) mm, rotated rx 180 ry 0 rz -80 deg; joints [-23.76, 59.979, 0, 82.056, 62.147, 109.896, -147.689]
  Call ExtruderHandler(155.587...: ExtruderHandler(155.58749)
  MoveL 151 to (-6.96, 20.32, 1.5) mm, rotated rx 180 ry 0 rz -100 deg; joints [-28.977, 56.923, 0, 89.737, 74.031, 100.392, -148.743]
  Call ExtruderHandler(13.33761)
  MoveL 152 to (-3.71, 20.89, 1.5) mm, rotated rx 180 ry 0 rz -100 deg; joints [-29.216, 56.706, 0, 90.299, 73.764, 100.422, -149.116]
  Call ExtruderHandler(141.783...: ExtruderHandler(141.78311)
  MoveL 153 to (21.05, -3.88, 1.5) mm, rotated rx -180 ry 0 rz -100 deg; joints [-28.038, 54.001, 0, 97.44, 74.09, 98.614, -153.269]
  Call ExtruderHandler(15.45103)
  MoveL 154 to (21.05, -0.06, 1.5) mm, rotated rx 180 ry 0 rz -100 deg; joints [-28.453, 54.14, 0, 97.066, 73.752, 98.87, -153.096]
  Call ExtruderHandler(121.804...: ExtruderHandler(121.80441)
  MoveL 155 to (-0.22, 21.22, 1.5) mm, rotated rx 180 ry 0 rz -100 deg; joints [-29.447, 56.462, 0, 90.928, 73.495, 100.433, -149.528]
  Call ExtruderHandler(19.04808)
  MoveL 156 to (4.41, 20.4, 1.5) mm, rotated rx -180 ry 0 rz -100 deg; joints [-29.63, 56.092, 0, 91.89, 73.231, 100.357, -150.134]
  Call ExtruderHandler(91.11339)
  MoveL 157 to (20.32, 4.48, 1.5) mm, rotated rx 180 ry 0 rz -100 deg; joints [-28.9, 54.358, 0, 96.481, 73.407, 99.181, -152.801]
  Call ExtruderHandler(19.96169)
  MoveL 158 to (18.64, 9.12, 1.5) mm, rotated rx 180 ry 0 rz -100 deg; joints [-29.294, 54.648, 0, 95.703, 73.132, 99.507, -152.385]
  Call ExtruderHandler(28.56215)
  MoveL 159 to (14.1, 14.52, 1.5) mm, rotated rx 180 ry 0 rz -100 deg; joints [-29.592, 55.17, 0, 94.313, 73.008, 99.903, -151.586]
  Call ExtruderHandler(11.93189)
  MoveL 160 to (12.02, 16.61, 1.5) mm, rotated rx 180 ry 0 rz -100 deg; joints [-29.686, 55.398, 0, 93.71, 72.988, 100.058, -151.236]
  Call MCodeHandler(104)
  Set speed (130.0 mm/s)
  MoveL 161 to (12.02, 16.61, 2.5) mm, rotated rx 180 ry 0 rz -100 deg; joints [-29.686, 55.26, 0, 93.758, 73.003, 100.085, -151.15]
  Call ExtruderHandler(-14.137...: ExtruderHandler(-14.13717)
  Set speed (40.0 mm/s)
  MoveL 162 to (12.02, 16.61, 2.5) mm, rotated rx 180 ry 0 rz -100 deg; joints [-29.686, 55.26, 0, 93.758, 73.003, 100.085, -151.15]
  Set speed (130.0 mm/s)
  MoveL 163 to (3.86, -25.06, 2.5) mm, rotated rx 180 ry 0 rz -80 deg; joints [-21.299, 60.646, 0, 80.156, 64.704, 109.074, -145.792]
  Call ExtruderHandler(14.13717)
  Set speed (40.0 mm/s)
  MoveL 164 to (3.86, -25.06, 2.5) mm, rotated rx 180 ry 0 rz -80 deg; joints [-21.299, 60.646, 0, 80.156, 64.704, 109.074, -145.792]
  Set speed (60.0 mm/s)
  MoveL 165 to (3.86, -25.06, 2.5) mm, rotated rx 180 ry 0 rz -80 deg; joints [-21.299, 60.646, 0, 80.156, 64.704, 109.074, -145.792]
  Call ExtruderHandler(8.87492)
  MoveL 166 to (8.8, -24.19, 2.5) mm, rotated rx 180 ry 0 rz -80 deg; joints [-21.577, 60.219, 0, 81.189, 64.273, 108.971, -146.45]
  Call ExtruderHandler(15.79840)
  MoveL 167 to (16.55, -19.72, 2.5) mm, rotated rx 180 ry 0 rz -80 deg; joints [-22.333, 59.682, 0, 82.499, 63.369, 109.049, -147.403]
  Call ExtruderHandler(15.79840)
  MoveL 168 to (22.29, -12.87, 2.5) mm, rotated rx 180 ry 0 rz -80 deg; joints [-23.255, 59.432, 0, 83.121, 62.434, 109.382, -148.024]
  Call ExtruderHandler(15.79840)
  MoveL 169 to (25.35, -4.47, 2.5) mm, rotated rx 180 ry 0 rz -80 deg; joints [-24.221, 59.493, 0, 82.982, 61.593, 109.937, -148.244]
  Call ExtruderHandler(15.79840)
  MoveL 170 to (25.35, 4.47, 2.5) mm, rotated rx 180 ry 0 rz -100 deg; joints [-29.199, 53.883, 0, 97.44, 73.064, 99.18, -153.314]
  Call ExtruderHandler(15.79841)
  MoveL 171 to (22.29, 12.87, 2.5) mm, rotated rx 180 ry 0 rz -100 deg; joints [-29.911, 54.409, 0, 96.027, 72.566, 99.773, -152.558]
  Call ExtruderHandler(15.79840)
  MoveL 172 to (16.55, 19.72, 2.5) mm, rotated rx 180 ry 0 rz -100 deg; joints [-30.278, 55.074, 0, 94.259, 72.425, 100.281, -151.547]
  Call ExtruderHandler(15.79840)
  MoveL 173 to (8.8, 24.19, 2.5) mm, rotated rx -180 ry 0 rz -100 deg; joints [-30.273, 55.801, 0, 92.35, 72.637, 100.633, -150.4]
  Call ExtruderHandler(15.79840)
  MoveL 174 to (0, 25.74, 2.5) mm, rotated rx 180 ry 0 rz -100 deg; joints [-29.915, 56.504, 0, 90.528, 73.152, 100.779, -149.254]
  Call ExtruderHandler(15.79840)
  MoveL 175 to (-8.8, 24.19, 2.5) mm, rotated rx 180 ry 0 rz -100 deg; joints [-29.262, 57.095, 0, 89.011, 73.885, 100.696, -148.246]
  Call ExtruderHandler(15.79841)
  MoveL 176 to (-16.55, 19.72, 2.5) mm, rotated rx -180 ry 0 rz -100 deg; joints [-28.395, 57.498, 0, 87.981, 74.739, 100.397, -147.497]
  Call ExtruderHandler(15.79840)
  MoveL 177 to (-22.29, 12.87, 2.5) mm, rotated rx 180 ry 0 rz -100 deg; joints [-27.41, 57.659, 0, 87.563, 75.62, 99.921, -147.099]
  Call ExtruderHandler(15.79840)
  MoveL 178 to (-25.35, 4.47, 2.5) mm, rotated rx 180 ry 0 rz -100 deg; joints [-26.411, 57.557, 0, 87.806, 76.441, 99.335, -147.099]
  Call ExtruderHandler(15.79840)
  MoveL 179 to (-25.35, -4.47, 2.5) mm, rotated rx 180 ry 0 rz -100 deg; joints [-25.501, 57.205, 0, 88.683, 77.129, 98.715, -147.498]
  Call ExtruderHandler(15.79840)
  MoveL 180 to (-22.29, -12.87, 2.5) mm, rotated rx 180 ry 0 rz -100 deg; joints [-24.781, 56.65, 0, 90.086, 77.619, 98.14, -148.246]
  Call ExtruderHandler(15.79840)
  MoveL 181 to (-16.55, -19.72, 2.5) mm, rotated rx 180 ry 0 rz -100 deg; joints [-24.335, 55.964, 0, 91.847, 77.855, 97.676, -149.255]
  Call ExtruderHandler(15.79841)
  MoveL 182 to (-8.8, -24.19, 2.5) mm, rotated rx -180 ry 0 rz -80 deg; joints [-20.907, 61.895, 0, 77.17, 65.594, 109.575, -144.009]
  Call ExtruderHandler(15.79840)
  MoveL 183 to (0, -25.74, 2.5) mm, rotated rx 180 ry 0 rz -80 deg; joints [-21.085, 60.985, 0, 79.341, 65.039, 109.153, -145.275]
  Call ExtruderHandler(6.52586)
  MoveL 184 to (3.64, -25.1, 2.5) mm, rotated rx 180 ry 0 rz -80 deg; joints [-21.287, 60.665, 0, 80.11, 64.723, 109.079, -145.763]
  Set speed (130.0 mm/s)
  MoveL 185 to (4.17, -26.8, 2.5) mm, rotated rx -180 ry 0 rz -80 deg; joints [-21.139, 60.553, 0, 80.378, 64.803, 108.928, -145.87]
  Set speed (60.0 mm/s)
  MoveL 186 to (4.17, -26.8, 2.5) mm, rotated rx -180 ry 0 rz -80 deg; joints [-21.139, 60.553, 0, 80.378, 64.803, 108.928, -145.87]
  Call ExtruderHandler(9.42556)
  MoveL 187 to (9.42, -25.88, 2.5) mm, rotated rx 180 ry 0 rz -80 deg; joints [-21.434, 60.101, 0, 81.474, 64.347, 108.818, -146.568]
  Call ExtruderHandler(16.89967)
  MoveL 188 to (17.7, -21.09, 2.5) mm, rotated rx 180 ry 0 rz -80 deg; joints [-22.242, 59.528, 0, 82.875, 63.381, 108.901, -147.585]
  Call ExtruderHandler(16.89967)
  MoveL 189 to (23.85, -13.77, 2.5) mm, rotated rx 180 ry 0 rz -80 deg; joints [-23.232, 59.261, 0, 83.539, 62.377, 109.255, -148.249]
  Call ExtruderHandler(16.89967)
  MoveL 190 to (27.12, -4.78, 2.5) mm, rotated rx 180 ry 0 rz -80 deg; joints [-24.269, 59.326, 0, 83.391, 61.473, 109.847, -148.485]
  Call ExtruderHandler(16.89967)
  MoveL 191 to (27.12, 4.78, 2.5) mm, rotated rx -180 ry 0 rz -100 deg; joints [-29.34, 53.779, 0, 97.725, 72.909, 99.191, -153.51]
  Call ExtruderHandler(16.89968)
  MoveL 192 to (23.85, 13.77, 2.5) mm, rotated rx -180 ry 0 rz -100 deg; joints [-30.1, 54.341, 0, 96.213, 72.377, 99.826, -152.701]
  Call ExtruderHandler(16.89967)
  MoveL 193 to (17.7, 21.09, 2.5) mm, rotated rx -180 ry 0 rz -100 deg; joints [-30.49, 55.051, 0, 94.322, 72.229, 100.371, -151.619]
  Call ExtruderHandler(16.89967)
  MoveL 194 to (9.42, 25.88, 2.5) mm, rotated rx 180 ry 0 rz -100 deg; joints [-30.48, 55.83, 0, 92.28, 72.462, 100.75, -150.392]
  Call ExtruderHandler(16.89967)
  MoveL 195 to (0, 27.54, 2.5) mm, rotated rx 180 ry 0 rz -100 deg; joints [-30.095, 56.582, 0, 90.331, 73.018, 100.907, -149.167]
  Call ExtruderHandler(16.89967)
  MoveL 196 to (-9.42, 25.88, 2.5) mm, rotated rx -180 ry 0 rz -100 deg; joints [-29.395, 57.215, 0, 88.708, 73.804, 100.819, -148.088]
  Call ExtruderHandler(16.89967)
  MoveL 197 to (-17.7, 21.09, 2.5) mm, rotated rx 180 ry 0 rz -100 deg; joints [-28.469, 57.647, 0, 87.606, 74.716, 100.497, -147.287]
  Call ExtruderHandler(16.89967)
  MoveL 198 to (-23.85, 13.77, 2.5) mm, rotated rx 180 ry 0 rz -100 deg; joints [-27.419, 57.82, 0, 87.158, 75.653, 99.986, -146.861]
  Call ExtruderHandler(16.89967)
  MoveL 199 to (-27.12, 4.78, 2.5) mm, rotated rx 180 ry 0 rz -100 deg; joints [-26.354, 57.711, 0, 87.419, 76.526, 99.358, -146.862]
  Call ExtruderHandler(16.89967)
  MoveL 200 to (-27.12, -4.78, 2.5) mm, rotated rx 180 ry 0 rz -100 deg; joints [-25.383, 57.333, 0, 88.357, 77.259, 98.694, -147.288]
  Call ExtruderHandler(16.89967)
  MoveL 201 to (-23.85, -13.77, 2.5) mm, rotated rx -180 ry 0 rz -100 deg; joints [-24.613, 56.738, 0, 89.858, 77.782, 98.079, -148.088]
  Call ExtruderHandler(16.89967)
  MoveL 202 to (-17.7, -21.09, 2.5) mm, rotated rx -180 ry 0 rz -100 deg; joints [-24.134, 56.004, 0, 91.742, 78.037, 97.584, -149.168]
  Call ExtruderHandler(16.89967)
  MoveL 203 to (-9.42, -25.88, 2.5) mm, rotated rx -180 ry 0 rz -80 deg; joints [-20.721, 61.891, 0, 77.177, 65.751, 109.463, -143.959]
  Call ExtruderHandler(16.89967)
  MoveL 204 to (0, -27.54, 2.5) mm, rotated rx 180 ry 0 rz -80 deg; joints [-20.909, 60.918, 0, 79.498, 65.162, 109.013, -145.312]
  Call ExtruderHandler(7.07650)
  MoveL 205 to (3.94, -26.84, 2.5) mm, rotated rx -180 ry 0 rz -80 deg; joints [-21.127, 60.572, 0, 80.332, 64.822, 108.932, -145.841]
  Set speed (130.0 mm/s)
  MoveL 206 to (4.44, -28.38, 2.5) mm, rotated rx -180 ry 0 rz -80 deg; joints [-20.993, 60.469, 0, 80.578, 64.893, 108.795, -145.94]
  Set speed (30.0 mm/s)
  MoveL 207 to (4.44, -28.38, 2.5) mm, rotated rx -180 ry 0 rz -80 deg; joints [-20.993, 60.469, 0, 80.578, 64.893, 108.795, -145.94]
  Call ExtruderHandler(8.06137)
  MoveL 208 to (9.97, -27.4, 2.5) mm, rotated rx 180 ry 0 rz -80 deg; joints [-21.303, 59.994, 0, 81.731, 64.415, 108.68, -146.674]
  Call ExtruderHandler(14.53765)
  MoveL 209 to (18.74, -22.34, 2.5) mm, rotated rx 180 ry 0 rz -80 deg; joints [-22.16, 59.389, 0, 83.213, 63.393, 108.766, -147.75]
  Call ExtruderHandler(14.53764)
  MoveL 210 to (25.26, -14.58, 2.5) mm, rotated rx -180 ry 0 rz -80 deg; joints [-23.212, 59.107, 0, 83.916, 62.327, 109.14, -148.453]
  Call ExtruderHandler(14.53764)
  MoveL 211 to (28.72, -5.06, 2.5) mm, rotated rx 180 ry 0 rz -80 deg; joints [-24.313, 59.176, 0, 83.759, 61.365, 109.766, -148.702]
  Call ExtruderHandler(14.53764)
  MoveL 212 to (28.72, 5.06, 2.5) mm, rotated rx -180 ry 0 rz -100 deg; joints [-29.468, 53.686, 0, 97.983, 72.768, 99.201, -153.687]
  Call ExtruderHandler(14.53765)
  MoveL 213 to (25.26, 14.58, 2.5) mm, rotated rx 180 ry 0 rz -100 deg; joints [-30.272, 54.279, 0, 96.381, 72.205, 99.875, -152.83]
  Call ExtruderHandler(14.53764)
  MoveL 214 to (18.74, 22.34, 2.5) mm, rotated rx 180 ry 0 rz -100 deg; joints [-30.682, 55.031, 0, 94.378, 72.052, 100.453, -151.684]
  Call ExtruderHandler(14.53765)
  MoveL 215 to (9.97, 27.4, 2.5) mm, rotated rx 180 ry 0 rz -100 deg; joints [-30.668, 55.856, 0, 92.215, 72.304, 100.856, -150.385]
  Call ExtruderHandler(14.53764)
  MoveL 216 to (0, 29.16, 2.5) mm, rotated rx 180 ry 0 rz -100 deg; joints [-30.257, 56.653, 0, 90.151, 72.898, 101.023, -149.087]
  Call ExtruderHandler(14.53764)
  MoveL 217 to (-9.97, 27.4, 2.5) mm, rotated rx 180 ry 0 rz -100 deg; joints [-29.515, 57.325, 0, 88.433, 73.732, 100.93, -147.945]
  Call ExtruderHandler(14.53765)
  MoveL 218 to (-18.74, 22.34, 2.5) mm, rotated rx -180 ry 0 rz -100 deg; joints [-28.536, 57.783, 0, 87.265, 74.696, 100.588, -147.097]
  Call ExtruderHandler(14.53764)
  MoveL 219 to (-25.26, 14.58, 2.5) mm, rotated rx 180 ry 0 rz -100 deg; joints [-27.427, 57.967, 0, 86.791, 75.684, 100.046, -146.645]
  Call ExtruderHandler(14.53765)
  MoveL 220 to (-28.72, 5.06, 2.5) mm, rotated rx 180 ry 0 rz -100 deg; joints [-26.303, 57.851, 0, 87.067, 76.604, 99.379, -146.646]
  Call ExtruderHandler(14.53764)
  MoveL 221 to (-28.72, -5.06, 2.5) mm, rotated rx -180 ry 0 rz -100 deg; joints [-25.277, 57.45, 0, 88.061, 77.375, 98.675, -147.097]
  Call ExtruderHandler(14.53764)
  MoveL 222 to (-25.25, -14.58, 2.5) mm, rotated rx 180 ry 0 rz -100 deg; joints [-24.461, 56.819, 0, 89.651, 77.929, 98.024, -147.945]
  Call ExtruderHandler(14.53764)
  MoveL 223 to (-18.74, -22.34, 2.5) mm, rotated rx -180 ry 0 rz -100 deg; joints [-23.951, 56.04, 0, 91.645, 78.202, 97.501, -149.088]
  Call ExtruderHandler(14.53765)
  MoveL 224 to (-9.97, -27.4, 2.5) mm, rotated rx -180 ry 0 rz -80 deg; joints [-20.553, 61.889, 0, 77.182, 65.893, 109.362, -143.913]
  Call ExtruderHandler(14.53764)
  MoveL 225 to (0, -29.16, 2.5) mm, rotated rx -180 ry 0 rz -80 deg; joints [-20.748, 60.859, 0, 79.64, 65.275, 108.886, -145.345]
  Call ExtruderHandler(6.15330)
  MoveL 226 to (4.22, -28.42, 2.5) mm, rotated rx 180 ry 0 rz -80 deg; joints [-20.981, 60.489, 0, 80.532, 64.912, 108.8, -145.911]
  Set speed (130.0 mm/s)
  MoveL 227 to (5.07, -27.02, 2.5) mm, rotated rx 180 ry 0 rz -80 deg; joints [-21.152, 60.461, 0, 80.6, 64.751, 108.88, -145.998]
  Call ExtruderHandler(-14.137...: ExtruderHandler(-14.13717)
  Set speed (40.0 mm/s)
  MoveL 228 to (5.07, -27.02, 2.5) mm, rotated rx 180 ry 0 rz -80 deg; joints [-21.152, 60.461, 0, 80.6, 64.751, 108.88, -145.998]
  Set speed (130.0 mm/s)
  MoveL 229 to (16.08, -17.66, 2.5) mm, rotated rx -180 ry 0 rz -80 deg; joints [-22.519, 59.802, 0, 82.211, 63.257, 109.227, -147.297]
  Call ExtruderHandler(14.13717)
  Set speed (40.0 mm/s)
  MoveL 230 to (16.08, -17.66, 2.5) mm, rotated rx -180 ry 0 rz -80 deg; joints [-22.519, 59.802, 0, 82.211, 63.257, 109.227, -147.297]
  Set speed (15.0 mm/s)
  MoveL 231 to (16.08, -17.66, 2.5) mm, rotated rx -180 ry 0 rz -80 deg; joints [-22.519, 59.802, 0, 82.211, 63.257, 109.227, -147.297]
  Call ExtruderHandler(3.56995)
  MoveL 232 to (14.71, -19.03, 2.5) mm, rotated rx 180 ry 0 rz -80 deg; joints [-22.326, 59.874, 0, 82.034, 63.46, 109.168, -147.141]
  Call ExtruderHandler(13.01135)
  MoveL 233 to (8.56, -22.58, 2.5) mm, rotated rx 180 ry 0 rz -80 deg; joints [-21.728, 60.301, 0, 80.992, 64.177, 109.106, -146.384]
  Call ExtruderHandler(35.70966)
  MoveL 234 to (22.33, -8.82, 2.5) mm, rotated rx -180 ry 0 rz -80 deg; joints [-23.659, 59.586, 0, 82.747, 62.142, 109.701, -147.94]
  Call ExtruderHandler(7.96840)
  MoveL 235 to (23.81, -4.74, 2.5) mm, rotated rx -180 ry 0 rz -80 deg; joints [-24.127, 59.618, 0, 82.677, 61.736, 109.972, -148.046]
  Call ExtruderHandler(49.08270)
  MoveL 236 to (4.9, -23.65, 2.5) mm, rotated rx 180 ry 0 rz -80 deg; joints [-21.478, 60.601, 0, 80.266, 64.528, 109.149, -145.906]
  Call ExtruderHandler(5.87121)
  MoveL 237 to (1.75, -24.21, 2.5) mm, rotated rx 180 ry 0 rz -80 deg; joints [-21.302, 60.876, 0, 79.603, 64.802, 109.214, -145.484]
  Call ExtruderHandler(58.45567)
  MoveL 238 to (24.27, -1.68, 2.5) mm, rotated rx 180 ry 0 rz -100 deg; joints [-28.467, 53.726, 0, 97.857, 73.683, 98.77, -153.465]
  Call ExtruderHandler(4.76248)
  MoveL 239 to (24.27, 0.91, 2.5) mm, rotated rx 180 ry 0 rz -100 deg; joints [-28.75, 53.822, 0, 97.601, 73.453, 98.945, -153.347]
  Call ExtruderHandler(66.07486)
  MoveL 240 to (-1.19, -24.55, 2.5) mm, rotated rx 180 ry 0 rz -80 deg; joints [-21.157, 61.143, 0, 78.964, 65.046, 109.288, -145.085]
  Call ExtruderHandler(4.11106)
  MoveL 241 to (-3.4, -24.16, 2.5) mm, rotated rx 180 ry 0 rz -80 deg; joints [-21.112, 61.369, 0, 78.422, 65.185, 109.394, -144.769]
  Call ExtruderHandler(71.80046)
  MoveL 242 to (24.27, 3.51, 2.5) mm, rotated rx -180 ry 0 rz -100 deg; joints [-29.031, 53.918, 0, 97.342, 73.225, 99.121, -153.229]
  Call ExtruderHandler(2.45264)
  MoveL 243 to (24.27, 4.85, 2.5) mm, rotated rx 180 ry 0 rz -100 deg; joints [-29.175, 53.968, 0, 97.207, 73.108, 99.212, -153.167]
  Call ExtruderHandler(1.80216)
  MoveL 244 to (23.93, 5.77, 2.5) mm, rotated rx 180 ry 0 rz -100 deg; joints [-29.254, 54.026, 0, 97.053, 73.053, 99.276, -153.085]
  Call ExtruderHandler(76.65436)
  MoveL 245 to (-5.6, -23.77, 2.5) mm, rotated rx -180 ry 0 rz -80 deg; joints [-21.067, 61.598, 0, 77.878, 65.325, 109.5, -144.452]
  Call ExtruderHandler(4.11106)
  MoveL 246 to (-7.81, -23.38, 2.5) mm, rotated rx 180 ry 0 rz -80 deg; joints [-21.022, 61.828, 0, 77.33, 65.465, 109.606, -144.132]
  Call ExtruderHandler(80.58270)
  MoveL 247 to (23.24, 7.67, 2.5) mm, rotated rx 180 ry 0 rz -100 deg; joints [-29.416, 54.144, 0, 96.735, 72.938, 99.41, -152.914]
  Call ExtruderHandler(3.71572)
  MoveL 248 to (22.55, 9.57, 2.5) mm, rotated rx 180 ry 0 rz -100 deg; joints [-29.577, 54.263, 0, 96.415, 72.826, 99.544, -152.743]
  Call ExtruderHandler(83.76130)
  MoveL 249 to (-9.72, -22.7, 2.5) mm, rotated rx -180 ry 0 rz -80 deg; joints [-21.017, 62.043, 0, 76.82, 65.566, 109.724, -143.846]
  Call ExtruderHandler(3.48638)
  MoveL 250 to (-11.37, -21.75, 2.5) mm, rotated rx 180 ry 0 rz -80 deg; joints [-21.047, 62.243, 0, 76.347, 65.63, 109.855, -143.591]
  Call ExtruderHandler(86.23397)
  MoveL 251 to (21.86, 11.48, 2.5) mm, rotated rx 180 ry 0 rz -100 deg; joints [-29.737, 54.383, 0, 96.093, 72.715, 99.679, -152.571]
  Call ExtruderHandler(2.31299)
  MoveL 252 to (21.43, 12.66, 2.5) mm, rotated rx 180 ry 0 rz -100 deg; joints [-29.836, 54.459, 0, 95.892, 72.647, 99.763, -152.465]
  Call ExtruderHandler(1.27615)
  MoveL 253 to (20.98, 13.19, 2.5) mm, rotated rx -180 ry 0 rz -100 deg; joints [-29.865, 54.51, 0, 95.755, 72.635, 99.803, -152.386]
  Call ExtruderHandler(88.22505)
  MoveL 254 to (-13.02, -20.8, 2.5) mm, rotated rx 180 ry 0 rz -80 deg; joints [-21.078, 62.445, 0, 75.871, 65.694, 109.987, -143.334]
  Call ExtruderHandler(3.48638)
  MoveL 255 to (-14.66, -19.85, 2.5) mm, rotated rx -180 ry 0 rz -100 deg; joints [-24.412, 55.817, 0, 92.23, 77.758, 97.666, -149.496]
  Call ExtruderHandler(89.42201)
  MoveL 256 to (19.79, 14.6, 2.5) mm, rotated rx 180 ry 0 rz -100 deg; joints [-29.942, 54.646, 0, 95.393, 72.604, 99.907, -152.178]
  Call ExtruderHandler(3.38045)
  MoveL 257 to (18.61, 16.02, 2.5) mm, rotated rx 180 ry 0 rz -100 deg; joints [-30.018, 54.782, 0, 95.029, 72.574, 100.011, -151.97]
  Call ExtruderHandler(90.45458)
  MoveL 258 to (-16.24, -18.84, 2.5) mm, rotated rx -180 ry 0 rz -100 deg; joints [-24.444, 55.972, 0, 91.828, 77.763, 97.735, -149.256]
  Call ExtruderHandler(3.38045)
  MoveL 259 to (-17.43, -17.43, 2.5) mm, rotated rx 180 ry 0 rz -100 deg; joints [-24.536, 56.112, 0, 91.467, 77.713, 97.83, -149.049]
  Call ExtruderHandler(90.45458)
  MoveL 260 to (17.43, 17.43, 2.5) mm, rotated rx -180 ry 0 rz -100 deg; joints [-30.094, 54.92, 0, 94.664, 72.546, 100.116, -151.761]
  Call ExtruderHandler(3.38045)
  MoveL 261 to (16.24, 18.84, 2.5) mm, rotated rx 180 ry 0 rz -100 deg; joints [-30.169, 55.059, 0, 94.298, 72.518, 100.22, -151.552]
  Call ExtruderHandler(90.45457)
  MoveL 262 to (-18.61, -16.02, 2.5) mm, rotated rx 180 ry 0 rz -100 deg; joints [-24.628, 56.252, 0, 91.106, 77.664, 97.926, -148.841]
  Call ExtruderHandler(3.38045)
  MoveL 263 to (-19.79, -14.61, 2.5) mm, rotated rx -180 ry 0 rz -100 deg; joints [-24.72, 56.394, 0, 90.742, 77.616, 98.021, -148.633]
  Call ExtruderHandler(89.42203)
  MoveL 264 to (14.66, 19.85, 2.5) mm, rotated rx 180 ry 0 rz -100 deg; joints [-30.179, 55.21, 0, 93.9, 72.552, 100.299, -151.314]
  Call ExtruderHandler(3.48638)
  MoveL 265 to (13.02, 20.8, 2.5) mm, rotated rx -180 ry 0 rz -100 deg; joints [-30.178, 55.363, 0, 93.495, 72.596, 100.374, -151.071]
  Call ExtruderHandler(88.22506)
  MoveL 266 to (-20.98, -13.19, 2.5) mm, rotated rx 180 ry 0 rz -100 deg; joints [-24.81, 56.536, 0, 90.378, 77.569, 98.117, -148.425]
  Call ExtruderHandler(1.27618)
  MoveL 267 to (-21.43, -12.66, 2.5) mm, rotated rx 180 ry 0 rz -100 deg; joints [-24.845, 56.591, 0, 90.239, 77.552, 98.154, -148.346]
  Call ExtruderHandler(2.31297)
  MoveL 268 to (-21.86, -11.48, 2.5) mm, rotated rx 180 ry 0 rz -100 deg; joints [-24.947, 56.667, 0, 90.044, 77.481, 98.234, -148.241]
  Call ExtruderHandler(86.23399)
  MoveL 269 to (11.37, 21.75, 2.5) mm, rotated rx -180 ry 0 rz -100 deg; joints [-30.177, 55.518, 0, 93.09, 72.641, 100.449, -150.827]
  Call ExtruderHandler(3.48638)
  MoveL 270 to (9.72, 22.7, 2.5) mm, rotated rx 180 ry 0 rz -100 deg; joints [-30.176, 55.673, 0, 92.682, 72.686, 100.523, -150.582]
  Call ExtruderHandler(83.76132)
  MoveL 271 to (-22.55, -9.57, 2.5) mm, rotated rx 180 ry 0 rz -100 deg; joints [-25.112, 56.792, 0, 89.728, 77.368, 98.364, -148.072]
  Call ExtruderHandler(3.71572)
  MoveL 272 to (-23.24, -7.67, 2.5) mm, rotated rx -180 ry 0 rz -100 deg; joints [-25.275, 56.917, 0, 89.41, 77.257, 98.494, -147.903]
  Call ExtruderHandler(80.58272)
  MoveL 273 to (7.81, 23.38, 2.5) mm, rotated rx 180 ry 0 rz -100 deg; joints [-30.132, 55.838, 0, 92.253, 72.772, 100.58, -150.318]
  Call ExtruderHandler(4.11106)
  MoveL 274 to (5.6, 23.77, 2.5) mm, rotated rx 180 ry 0 rz -100 deg; joints [-30.042, 56.012, 0, 91.799, 72.901, 100.617, -150.032]
  Call ExtruderHandler(76.65439)
  MoveL 275 to (-23.93, -5.77, 2.5) mm, rotated rx 180 ry 0 rz -100 deg; joints [-25.437, 57.044, 0, 89.091, 77.147, 98.625, -147.733]
  Call ExtruderHandler(1.80217)
  MoveL 276 to (-24.27, -4.85, 2.5) mm, rotated rx 180 ry 0 rz -100 deg; joints [-25.516, 57.105, 0, 88.936, 77.094, 98.689, -147.65]
  Call ExtruderHandler(2.45262)
  MoveL 277 to (-24.27, -3.51, 2.5) mm, rotated rx -180 ry 0 rz -100 deg; joints [-25.653, 57.157, 0, 88.807, 76.989, 98.781, -147.592]
  Call ExtruderHandler(71.80049)
  MoveL 278 to (3.4, 24.16, 2.5) mm, rotated rx -180 ry 0 rz -100 deg; joints [-29.953, 56.188, 0, 91.342, 73.029, 100.653, -149.745]
  Call ExtruderHandler(4.11106)
  MoveL 279 to (1.19, 24.55, 2.5) mm, rotated rx 180 ry 0 rz -100 deg; joints [-29.864, 56.366, 0, 90.884, 73.157, 100.689, -149.457]
  Call ExtruderHandler(66.07489)
  MoveL 280 to (-24.27, -0.91, 2.5) mm, rotated rx -180 ry 0 rz -100 deg; joints [-25.918, 57.258, 0, 88.555, 76.787, 98.96, -147.477]
  Call ExtruderHandler(4.76249)
  MoveL 281 to (-24.27, 1.68, 2.5) mm, rotated rx 180 ry 0 rz -100 deg; joints [-26.182, 57.36, 0, 88.3, 76.587, 99.14, -147.361]
  Call ExtruderHandler(58.45570)
  MoveL 282 to (-1.75, 24.21, 2.5) mm, rotated rx -180 ry 0 rz -100 deg; joints [-29.661, 56.567, 0, 90.364, 73.391, 100.676, -149.114]
  Call ExtruderHandler(5.87120)
  MoveL 283 to (-4.9, 23.65, 2.5) mm, rotated rx 180 ry 0 rz -100 deg; joints [-29.427, 56.777, 0, 89.822, 73.654, 100.646, -148.754]
  Call ExtruderHandler(49.08277)
  MoveL 284 to (-23.81, 4.74, 2.5) mm, rotated rx 180 ry 0 rz -100 deg; joints [-26.515, 57.445, 0, 88.089, 76.326, 99.352, -147.282]
  Call ExtruderHandler(7.96838)
  MoveL 285 to (-22.32, 8.82, 2.5) mm, rotated rx -180 ry 0 rz -100 deg; joints [-27.002, 57.494, 0, 87.973, 75.924, 99.636, -147.282]
  Call ExtruderHandler(35.70982)
  MoveL 286 to (-8.57, 22.58, 2.5) mm, rotated rx 180 ry 0 rz -100 deg; joints [-29.115, 57.007, 0, 89.232, 73.988, 100.581, -148.353]
  Call ExtruderHandler(13.01135)
  MoveL 287 to (-14.71, 19.03, 2.5) mm, rotated rx 180 ry 0 rz -100 deg; joints [-28.425, 57.326, 0, 88.416, 74.667, 100.344, -147.76]
  Call ExtruderHandler(3.57040)
  MoveL 288 to (-16.08, 17.66, 2.5) mm, rotated rx 180 ry 0 rz -100 deg; joints [-28.214, 57.374, 0, 88.292, 74.86, 100.249, -147.653]
  Call ExtruderHandler(-14.137...: ExtruderHandler(-14.13717)
  Set speed (40.0 mm/s)
  MoveL 289 to (-16.08, 17.66, 2.5) mm, rotated rx 180 ry 0 rz -100 deg; joints [-28.214, 57.374, 0, 88.292, 74.86, 100.249, -147.653]
  MoveL 290 to (-16.08, 17.66, 2.5) mm, rotated rx 180 ry 0 rz -100 deg; joints [-28.214, 57.374, 0, 88.292, 74.86, 100.249, -147.653]
  MoveL 291 to (-16.08, 17.66, 152.5) mm, rotated rx 180 ry 0 rz -100 deg; joints [-28.306, 39.453, 0, 90.496, 78.094, 104.008, -132.039]
  Call MCodeHandler(104)
  Call MCodeHandler(84)
  Call MCodeHandler(140)
